FUNCTION_BLOCK FB_XPIM_States EXTENDS FB_PositionStateBase_WithPMPS
VAR_INPUT
    {attribute 'pytmc' := '
        pv: SET
        io: io
    '}
    enumSet: ENUM_XPIM_states;

    stOut: DUT_PositionState;
    stYag: DUT_PositionState;
    stDiamond: DUT_PositionState;
    stReticle: DUT_PositionState;

    bStatesLock: BOOL;
END_VAR
VAR_OUTPUT
    {attribute 'pytmc' := '
        pv: GET
        io: i
    '}
    enumGet: ENUM_XPIM_States;
END_VAR
VAR
    fbStateDefaults: FB_PositionState_Defaults;
    bXPIMInit: BOOL;
END_VAR
VAR CONSTANT
    fInDelta: LREAL := 2;
    fOutDelta: LREAL := 2;
    fInVelocity: LREAL := 1;
    fOutVelocity: LREAL := 1;
    fAccel: LREAL := 200;
    fOutDecel: LREAL := 25;
END_VAR

IF NOT bXPIMInit THEN
    bXPIMInit := TRUE;

    stOut.sName := 'OUT';
    fbStateDefaults(
        stPositionState:=stOut,
        fVeloDefault:=fOutVelocity,
        fDeltaDefault:=fOutDelta,
        fAccelDefault:=fAccel,
        fDecelDefault:=fOutDecel,
    );
    stOut.bMoveOk := TRUE;

    stYag.sName := 'YAG';
    fbStateDefaults(
        stPositionState:=stYag,
        fVeloDefault:=fInVelocity,
        fDeltaDefault:=fInDelta,
        fAccelDefault:=fAccel,
        fDecelDefault:=fAccel,
    );
    stYag.bMoveOk := TRUE;

    stDiamond.sName := 'DIAMOND';
    fbStateDefaults(
        stPositionState:=stDiamond,
        fVeloDefault:=fInVelocity,
        fDeltaDefault:=fInDelta,
        fAccelDefault:=fAccel,
        fDecelDefault:=fAccel,
    );
    stDiamond.bMoveOk := TRUE;

    stReticle.sName := 'RETICLE';
    fbStateDefaults(
        stPositionState:=stReticle,
        fVeloDefault:=fInVelocity,
        fDeltaDefault:=fInDelta,
        fAccelDefault:=fAccel,
        fDecelDefault:=fAccel,
    );
    stReticle.bMoveOk := TRUE;

    arrStates[1] := stOut;
    arrStates[2] := stYag;
    arrStates[3] := stDiamond;
    arrStates[4] := stReticle;
END_IF

setState := enumSet;
Exec();
enumGet := getState;
enumSet := setState;

END_FUNCTION_BLOCK

(* stored: Version 1.1.0.1
   POU FB_XPIM_States: Id {8c4640db-3bb7-4671-b4ea-e9d46c4b8221}, SpecialFunc None *)
